FUNCTION_BLOCK QUERY_STATION5
  {SET_ATTRIBUTE(OpcUa, SERVICE)}
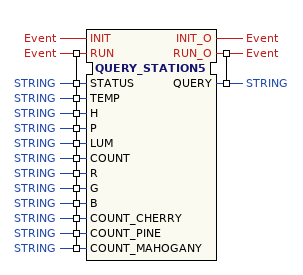
  EVENT_INPUT
    INIT;
    RUN WITH STATUS, TEMP, H, P, LUM, COUNT, R, G, B, COUNT_CHERRY, COUNT_PINE, COUNT_MAHOGANY; {SET_ATTRIBUTE(OpcUa, Method)}
  END_EVENT
  EVENT_OUTPUT
    INIT_O;
    RUN_O WITH QUERY;
  END_EVENT
  VAR_INPUT
    STATUS : STRING;
    TEMP : STRING;
    H : STRING;
    P : STRING;
    LUM : STRING;
    COUNT : STRING;
    R : STRING;
    G : STRING;
    B : STRING;
    COUNT_CHERRY : STRING;
    COUNT_PINE : STRING;
    COUNT_MAHOGANY : STRING;
  END_VAR
  VAR_OUTPUT
    QUERY : STRING;
  END_VAR
END_FUNCTION_BLOCK
